_CFC_ (* Continuous Function Chart, elements in execution order *)
#0 REAL_TO_TIME(SHU6_P2_P1_ZADER_Z_P1_OTKAZ)
#1 MUL(#0, 1000)
#2 delayFBC_P1 <= #1
#3 TON_P1_VKL_Leto:TON(IN: NOT SHU6_P2_P1_DO7, PT: T#43200s)
#4 OR(SHU6_P2_UST_ZIMA, SHU6_P2_Z_ZAM_SRAB, #3.Q)
#5 TON_P1_OTKL_Leto:TON(IN: SHU6_P2_P1_DO7, PT: T#10s)
#6 AND(SHU6_P2_UST_LETO, #5.Q)
#7 SR_P1:SR(SET1: #4, RESET: #6)
#8 SEL(SHU6_P2_P1_DI5_A, eHVACActuatorMode_Off_OP, eHVACActuatorMode_Auto_BMS)
#9 AND(SHU6_P2_P1_DI5_A, SHU6_P2_P1_DI7_RUN)
#10 fb_HVACMS_P1:FB_HVACMotor1Speed(eHVACDataSecurityType_Idle, FALSE, TRUE, #7.Q1, #8, NOT SHU6_P2_Z_P1_NPIT, #9, NOT SHU6_P2_Z_P1_OTKAZ, TRUE, TRUE, SHU6_P2_KV1_DI8, SHU6_P2_SB, startDelay_P1, stopDelay_P1, delayFBC_P1, feedbPT_P1, delayFBP_P1)
#11 SHU6_P2_P1_DO7 <= #10.out 1
#12 >(#10.out 8, 0)
#13 SHU6_P2_Z_P1_OTKAZ <= #12
#14 SHU6_P2_P1_DO5_ALM <= #12
_END_CFC_
END_PROGRAM

(* POU IM/MV2/MV2_1, CFC *)
PROGRAM MV2_1
VAR
	RS_M1: RS;

	startDelay_M1: TIME := T#0s;
	stopDelay_M1: TIME := T#0s;
	delayFBC_M1: TIME := T#30S;
	feedbPT_M1: TIME := T#120s;
	delayFBP_M1: TIME := T#30s;

	fb_HVACMS_M1: FB_HVACMotor1Speed;
	fb_HVACPIDC_M1: FB_HVACPIDCtrl;

	deadRange: REAL := 0.1;
	rKp: REAL := 1;
	tTi: TIME;
	tTv: TIME := T#0s;
	tTd: TIME := T#0s;
	direction: BOOL;
	rYMin: REAL;
	Dint_Ti: DINT;
	set: BOOL;
	reset: BOOL;
	resetContr: BOOL;
	SR_VKL: SR;
	TON_PUSK:TON;
	RT_PUSK : R_TRIG;
	TON_MV2_OTKAZ: TON;
	TON_NV2_OTKAZ: TON;
END_VAR
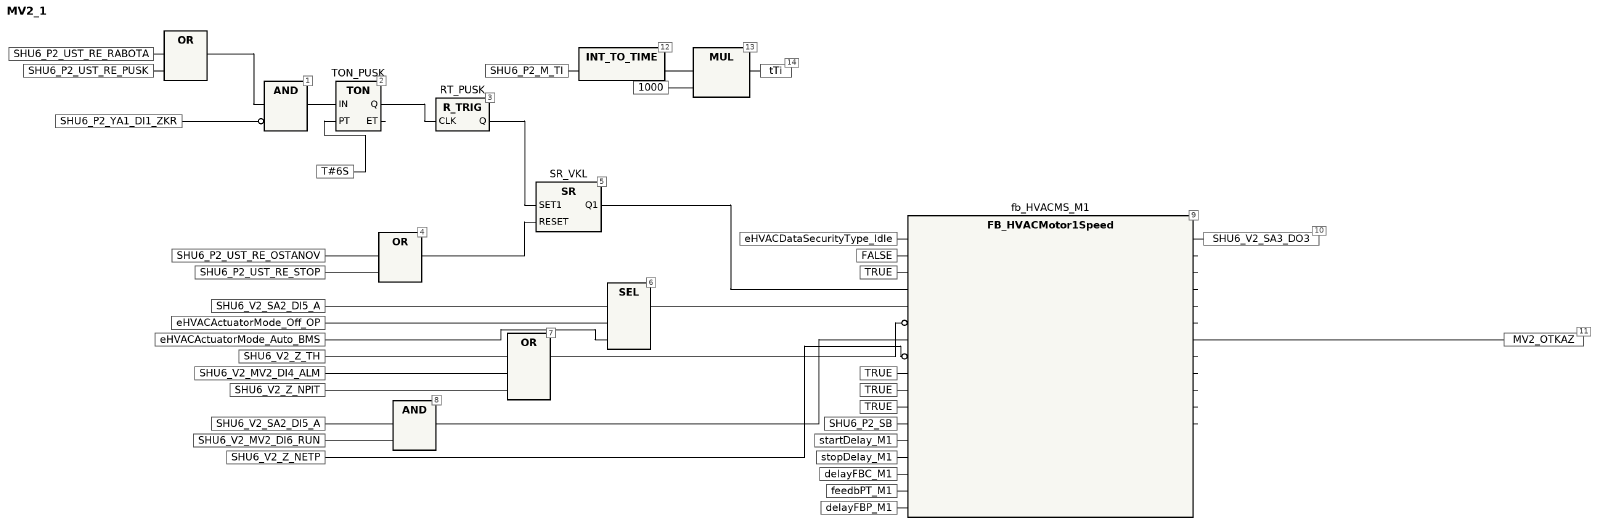
_CFC_ (* Continuous Function Chart, elements in execution order *)
#0 OR(SHU6_P2_UST_RE_RABOTA, SHU6_P2_UST_RE_PUSK)
#1 AND(#0, NOT SHU6_P2_YA1_DI1_ZKR)
#2 TON_PUSK:TON(IN: #1, PT: T#6S)
#3 RT_PUSK:R_TRIG(CLK: #2.Q)
#4 OR(SHU6_P2_UST_RE_OSTANOV, SHU6_P2_UST_RE_STOP)
#5 SR_VKL:SR(SET1: #3.Q, RESET: #4)
#6 SEL(SHU6_V2_SA2_DI5_A, eHVACActuatorMode_Off_OP, eHVACActuatorMode_Auto_BMS)
#7 OR(SHU6_V2_Z_TH, SHU6_V2_MV2_DI4_ALM, SHU6_V2_Z_NPIT)
#8 AND(SHU6_V2_SA2_DI5_A, SHU6_V2_MV2_DI6_RUN)
#9 fb_HVACMS_M1:FB_HVACMotor1Speed(eHVACDataSecurityType_Idle, FALSE, TRUE, #5.Q1, #6, NOT #7, #8, NOT SHU6_V2_Z_NETP, TRUE, TRUE, TRUE, SHU6_P2_SB, startDelay_M1, stopDelay_M1, delayFBC_M1, feedbPT_M1, delayFBP_M1)
#10 SHU6_V2_SA3_DO3 <= #9.out 1
#11 MV2_OTKAZ <= #9.out 7
#12 INT_TO_TIME(SHU6_P2_M_TI)
#13 MUL(#12, 1000)
#14 tTi <= #13
_END_CFC_
END_PROGRAM

(* POU IM/razr_pusk, CFC *)
PROGRAM razr_pusk
VAR
END_VAR
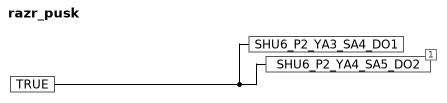
_CFC_ (* Continuous Function Chart, elements in execution order *)
#0 SHU6_P2_YA3_SA4_DO1 <= TRUE
#1 SHU6_P2_YA4_SA5_DO2 <= TRUE
_END_CFC_
(* the same logic as Structured Text *)
SHU6_P2_YA3_SA4_DO1 := TRUE;
SHU6_P2_YA4_SA5_DO2 := TRUE;
END_PROGRAM

(* POU IM/YA1_Upr, CFC *)
PROGRAM YA1_Upr
VAR
	RS_YA2_Open: RS;
	RT_Pusk: R_TRIG;
	RT_OSTANOV: R_TRIG;
	fb_HVACPA: FB_HVAC2PointActuator;

	stokeTime: TIME;
	enableLimitSwitch: BOOL := TRUE;
	FT_PCH_OTKL: R_TRIG;
	TON_PCH_OTKL: TON;
	ZADERJ_SHOD_YA2: TON;
	TON_OTK_MV: TON;
END_VAR
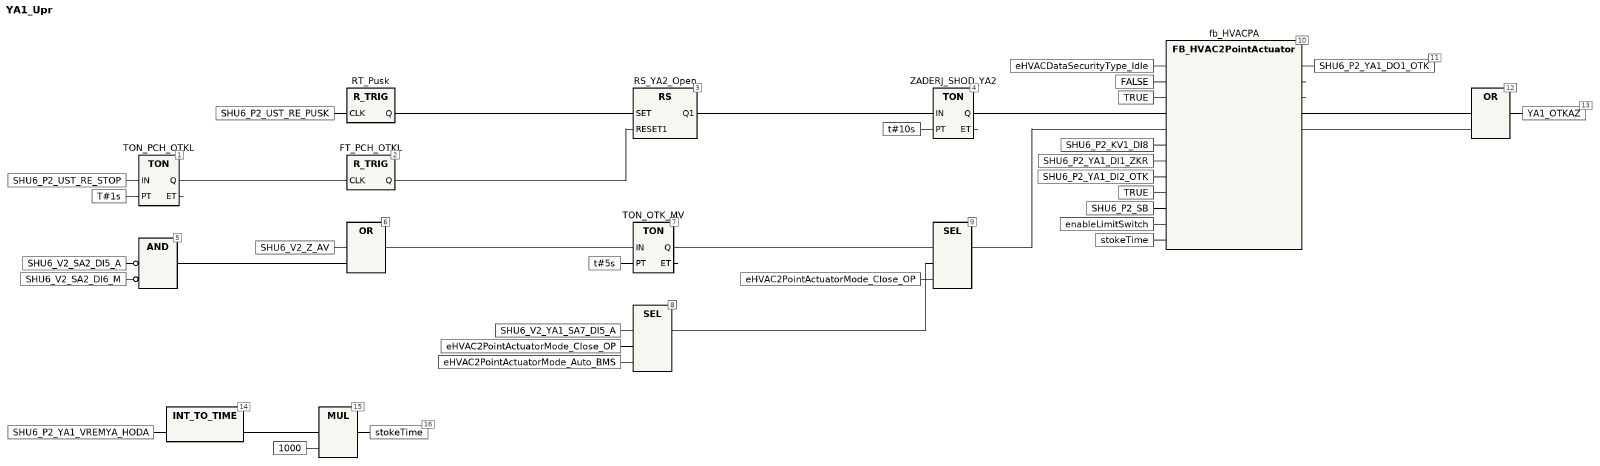
_CFC_ (* Continuous Function Chart, elements in execution order *)
#0 RT_Pusk:R_TRIG(CLK: SHU6_P2_UST_RE_PUSK)
#1 TON_PCH_OTKL:TON(IN: SHU6_P2_UST_RE_STOP, PT: T#1s)
#2 FT_PCH_OTKL:R_TRIG(CLK: #1.Q)
#3 RS_YA2_Open:RS(SET: #0.Q, RESET1: #2.Q)
#4 ZADERJ_SHOD_YA2:TON(IN: #3.Q1, PT: t#10s)
#5 AND(NOT SHU6_V2_SA2_DI5_A, NOT SHU6_V2_SA2_DI6_M)
#6 OR(SHU6_V2_Z_AV, #5)
#7 TON_OTK_MV:TON(IN: #6, PT: t#5s)
#8 SEL(SHU6_V2_YA1_SA7_DI5_A, eHVAC2PointActuatorMode_Close_OP, eHVAC2PointActuatorMode_Auto_BMS)
#9 SEL(#7.Q, #8, eHVAC2PointActuatorMode_Close_OP)
#10 fb_HVACPA:FB_HVAC2PointActuator(eHVACDataSecurityType_Idle, FALSE, TRUE, #4.Q, #9, SHU6_P2_KV1_DI8, SHU6_P2_YA1_DI1_ZKR, SHU6_P2_YA1_DI2_OTK, TRUE, SHU6_P2_SB, enableLimitSwitch, stokeTime)
#11 SHU6_P2_YA1_DO1_OTK <= #10.out 1
#12 OR(#10.out 4, #10.out 5)
#13 YA1_OTKAZ <= #12
#14 INT_TO_TIME(SHU6_P2_YA1_VREMYA_HODA)
#15 MUL(#14, 1000)
#16 stokeTime <= #15
_END_CFC_
END_PROGRAM

(* POU IM/YA2_Upr, CFC *)
PROGRAM YA2_Upr
VAR
	RS_YA2_Open: RS;
	RT_Pusk: R_TRIG;
	RT_OSTANOV: R_TRIG;
	fb_HVACPA: FB_HVAC2PointActuator;

	stokeTime: TIME;
	enableLimitSwitch: BOOL := TRUE;
	FT_PCH_OTKL: R_TRIG;
	TON_PCH_OTKL: TON;
	ZADERJ_SHOD_YA2: TON;
	TON_YA2_Z_ZAM_TE4: TON;
	TON_OTK_MV:TON;
END_VAR
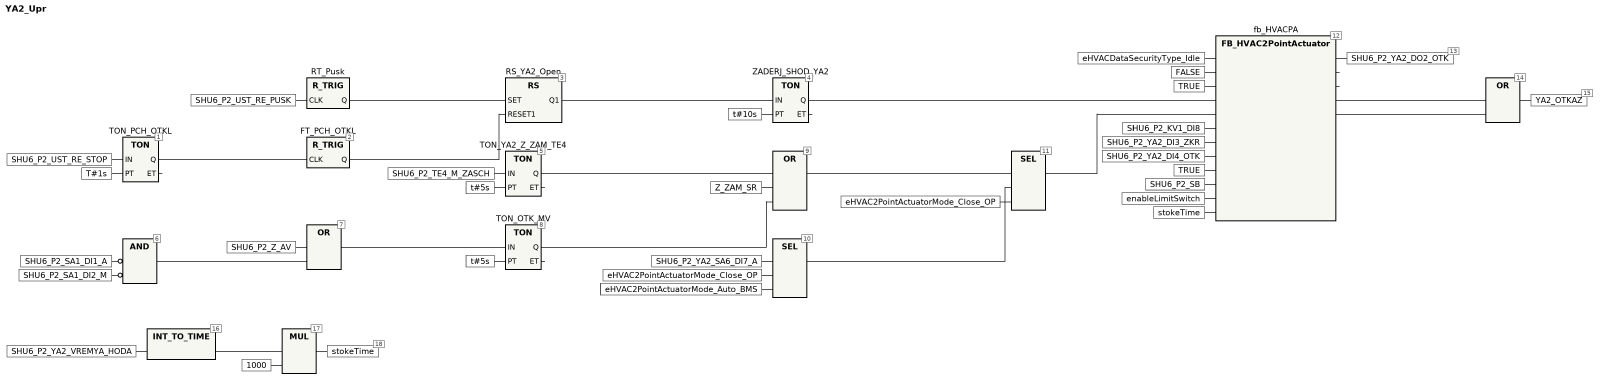
